// TIA Portal V20 export
DATA_BLOCK "BK22"   // DB269
// stored: MemoryReserve 100
   VAR
      "X10-1 INS TRANSFER P&P2 Y-AXIS LIMIT SENSOR(-)" : Bool;
      "X11-1 INS TRANSFER P&P2 Y-AXIS LIMIT SENSOR(+)" : Bool;
      "X12-1 INS TRANSFER P&P2 Z-AXIS LIMIT SENSOR(-)" : Bool;
      "X13-1 INS TRANSFER P&P2 Z-AXIS LIMIT SENSOR(+)" : Bool;
      "X14-1 INS TRANSFER P&P2 CLAMP OPEN SENSOR" : Bool;
      "X15-1 INS TRANSFER P&P2 CLAMP STACK DETECT SENSOR" : Bool;
      "X16-1 INS TRANSFER P&P2 Z-AXIS SAFETY PIN LOADING SENSOR" : Bool;
      "X17-1 SPARE" : Bool;
      "X10-2 INS TRANSFER P&P2 Y-AXIS HOMING SENSOR" : Bool;
      "X11-2 SPARE" : Bool;
      "X12-2 PROCESS P&P Z-AXIS HEAD2 HOMING SENSOR" : Bool;
      "X13-2 SPARE" : Bool;
      "X14-2 INS TRANSFER P&P2 CLAMP CLOSE SENSOR" : Bool;
      "X15-2 INS TRANSFER P&P2 CLAMP OPEN/CLOSE PRESSURE SENSOR" : Bool;
      "X16-2 SPARE" : Bool;
      "X17-2 SPARE" : Bool;
   END_VAR
BEGIN
END_DATA_BLOCK
